FUNCTION_BLOCK ModbusWriteWord EXTENDS ModbusIo
VAR_INPUT
	Value: WORD;
END_VAR
VAR_OUTPUT
END_VAR
VAR
END_VAR

SUPER^();

END_FUNCTION_BLOCK

(* stored: Version 1.1.0.1, ProductVersion 3.1.4024.2
   POU ModbusWriteWord: Id {53d5e34b-aeae-47d4-a08b-e0c8ea184e2e}, SpecialFunc None *)
